// TIA Portal V17 export
// export: Created 2024-09-02T12:50:31.1175098Z, ExportSetting WithDefaults, DisplayName Totally Integrated Automation Portal, DisplayVersion V17, DisplayName TIA Portal Openness, DisplayVersion V17, DisplayName TIA Portal Version Control Interface, DisplayVersion V17, DisplayName STEP 7 Professional, DisplayVersion V17, DisplayName STEP 7 Safety, DisplayVersion V17, DisplayName WinCC Professional, DisplayVersion V17
TYPE "TypeSKS_Desutter"
// stored: IsFailsafeCompliant false
   STRUCT
      "A" : Struct
         StartPRG : Array[0..20] of Bool;
         Acknowledge : Bool;
         Reset_outputs : Bool;
         Start_active : Bool;
         Start_active_fp : Bool;
         Start_unscrewing : Bool;
         Retry_activ : Bool;
         Retry_activ_fp : Bool;
         Start_timer_screwing { S7_SetPoint := 'True'} : IEC_TIMER;
         Start_timer_unscrewing { S7_SetPoint := 'True'} : IEC_TIMER;
      END_STRUCT;
      H : Struct
         StartPRG : Array[0..20] of Bool;
         Acknowledge : Bool;
         Reset_outputs : Bool;
         Start_active : Bool;
         Start_unscrewing : Bool;
      END_STRUCT;
   END_STRUCT;
END_TYPE
